TYPE ST_HW_InputsRejectPanel :
STRUCT
	RejectBtnEnable						: BOOL;                  //  RejectBtnEnable Signal To change colour of button after touch on reject panel
    ProfileBtnEnable					: BOOL;                  //  ProfileBtnEnable Signal To change colour of button after touch on reject panel
	WrapperBtnEnable					: BOOL;  				 //  WrapperBtnEnable Signal To change colour of button after touch on reject panel
	DepallatizerBtnEnable   			: BOOL; 				 //  DepallatizerBtnEnable Signal To change colour of button after touch on reject panel
END_STRUCT
END_TYPE

(* stored: Version 1.1.0.1, ProductVersion 3.1.4022.12
   DUT ST_HW_InputsRejectPanel: Id {80133d0d-e61b-44f9-a280-f890defd5506} *)
